
// ===== library: MasterCopy "BVS_Sensor" =====

FUNCTION_BLOCK "BVS_Sensor"   // FB52, SCL
TITLE = BVS_ID
{ S7_Optimized_Access := 'TRUE' }
AUTHOR : PD-ILS
FAMILY : Balluff
VERSION : 1.1
// Functionblock for BVS ID and BVS VS.
// Compatible with Profinet and IO-Link version.
   VAR_INPUT
      Init : Bool;   // Internal reset and initailisation of FB
      CommandStart : Bool;   // Start BVS command
      BVS_ResetError : Bool;   // Reset BVS errors
      BVS_Trigger : Bool;   // Trigger BVS
      Get_Results : Bool;   // Get BVS results
      HW_LADDR : HW_SUBMODULE;   // BVS hardware address
      Command : Int;   // 1=SwitchApp; 2=GetApp; 3=GetResult; 4=SetInput
      DB_Send : Int;   // Data block with BVS send data
      Offset_DBSend : Int;   // Offset send data
      DB_Receive : Int;   // Data block with BVS receive data
      Offset_DBReceive : Int;   // Offset receive data
      Data_Length : Int;   // Data length for set commando
      WD_Time : Time := T#120000ms;   // Watchdog of commandos
      PILen : UInt := 32;   // Input process data length
      PQLen : UInt := 32;   // Output process data length
   END_VAR
   VAR_OUTPUT
      Ready : Bool;   // Comamnd ready and FB ready
      BVS_WaitForTrigger : Bool;   // BVS waiting for Trigger
      BVS_ResultDataAvailable : Bool;   // BVS result ready
      BVS_Ready : Bool;   // BVS ready
      BVS_DeviceLocked : Bool;   // BVS is locked
      BVS_TriggerOverflowError : Bool;   // BVS warning overtriggerd
      BVS_ResultDataError : Bool;   // BVS warning result data error
      BVS_ReportError : Bool;   // BVS warning report error
      BVS_InputDataError : Bool;   // BVS warning input data error
      BVS_SystemError : Bool;   // BVS warning system error
      Error : Bool;   // Command or BVS Error
      ErrorNumber : Word;   // Error number
      ReceivedLength : Int;   // BVS received result buffer length
   END_VAR
   VAR
      PointerByte : Int;   // Pointer byte
      LengthByte : Int;   // Number of byte for set/get commando
      BytePerPageIn : Int;   // User bytes per page Out
      BytePerPageOut : Int;   // User bytes per page In
      TotalByte : Int;   // Over all byte data to be set/get
      LengOverhead : Int;   // Overhead length for get command
      StDataOffset : Int;   // Start Data Offset for set command
      HW_Init : Bool;   // Hardware adresses initialized
      GetCommandActive : Bool;   // Get commado activ
      SetCommandActive : Bool;   // Set commando active
      GComSend : Bool;   // Get Commando send
      ComDatEnd : Bool;   // Comand data transfered
      ToggleOld : Bool;   // Toggle bit last cycle
      FirstCycle : Bool;   // First command cycle
      IMP_Start : Bool;   // Rising edge Start
      IMP_ResetError : Bool;   // Rising edge Reset
      Cam_Reset : Bool;   // Start BVS reset
      ErrorIn : Bool;   // Error bit intern
      WD_TimerIn : Bool;   // Watchdog timer input
      WD_TimerQ : Bool;   // Watchdog timer output
      CO_WaitForTrigger : Bool;   // CAM Out - PLC In waiting for trigger BasAd[50]
      CO_ResultDataAvailable : Bool;   // CAM Out - PLC In result ready
      CO_R02 : Bool;   // CAM Out - PLC In reserved
      CO_R03 : Bool;   // CAM Out - PLC In simulation mode activated
      CO_R04 : Bool;   // CAM Out - PLC In reserved
      CO_Ready : Bool;   // CAM Out - PLC In ready
      CO_R06 : Bool;   // CAM Out - PLC In reserved
      CO_DeviceLocked : Bool;   // CAM Out - PLC In device locked
      CO_TriggerOverflow : Bool;   // CAM Out - PLC In error trigger overflow
      CO_ResultDataError : Bool;   // CAM Out - PLC In result data overwitten
      CO_ReportError : Bool;   // CAM Out - PLC In ftp report error
      CO_R13 : Bool;   // CAM Out - PLC In reserved
      CO_InputDataError : Bool;   // CAM Out - PLC Input data error
      CO_R15 : Bool;   // CAM Out - PLC In reserved
      CO_R16 : Bool;   // CAM Out - PLC In reserved
      CO_SystemError : Bool;   // CAM Out - PLC In system error
      CO_R20 : Bool;   // CAM Out - PLC In reserved
      CO_JobStartAA : Bool;   // CAM Out - PLC In job start
      CO_JobEndAE : Bool;   // CAM Out - PLC In job end
      CO_JobErrorAF : Bool;   // CAM Out - PLC In job error
      CO_R24 : Bool;   // CAM Out - PLC In reserved
      CO_ToggleOut : Bool;   // CAM Out - PLC In toggle out
      CO_OutArea : Array[0..#OutBuSi] of Byte;   // CAM Out - PLC In data area
      CI_AV_JobStart : Bool;   // PLC Out - CAM In job start
      CI_Trigger : Bool;   // PLC Out - CAM In trigger
      CI_ResetError : Bool;   // PLC Out - CAM In reset error
      CI_R03 : Bool;   // PLC Out - CAM In reserved
      CI_R04 : Bool;   // PLC Out - CAM In reserved
      CI_R05 : Bool;   // PLC Out - CAM In reserved
      CI_ToggleIn : Bool;   // PLC Out - CAM In toggle in
      CI_R07 : Bool;   // PLC Out - CAM In reserved
      CI_InLengInt : Int;   // PLC Out - CAM In length int
      CI_InArea : Array[0..#InBuSi] of Byte;   // PLC Out - CAM In input area
      OldCyComState : Word;   // Commando state last cycle
      WD_Timer : TON_TIME;   // Watchdog timer TON
      PIaddr : UDInt;   // Input address
      PIcount : UInt;   // Input length
      PQaddr : UDInt;   // Output address
      PQcount : UInt;   // Output address
      RetVal_ModulDiag : Int;   // Return value modul diagnosis
      RetVal_RD_Addr : Int;   // Return value read address
      RetVal_RD_DP : Int;   // Return value read input data
      RetVal_WR_DP : Int;   // Return value write output data
      RetVal_Get_ErrID : Word;   // Return value get error ID
      R_TRIG_ResetError : R_TRIG;   // R Trigger reset warning
      R_TRIG_CamTrg : R_TRIG;   // R Trigger BVS trigger
      R_TRIG_Start : R_TRIG;   // R Trigger BVS start
      ErrorCode : DWord;   // Internal BVS error code
      CNT_Diag : UInt;   // CNT_Modul Diag
      Diag_Out : DWord;   // Modul Diag
   END_VAR
   VAR_TEMP
      tError : Word;   // temp error buffer
      tLoop : DInt;   // temp loopcounter
   END_VAR
   VAR CONSTANT
      InBuSi : Int := 127;   // maximum size input buffer
      OutBuSi : Int := 127;   // maximum size output buffer
      ST_DATOFFSET : Int := 3;   // First DataOffset for set commands
   END_VAR
BEGIN
   //=============================================================================
   //Balluff GmbH
   //(c)Copyright (2024) All Rights Reserved
   //-----------------------------------------------------------------------------
   //Library: BalluffVision
   //Tested with: CPU 1214C V4.1
   //Engineering: TIA Portal V13 SP1 
   //Restrictions: -
   //Requirements: PLC (S7-1200 / S7-1500)
   //Functionality: Boolean BVS functions, BVS Commandos
   //-----------------------------------------------------------------------------
   //Change log table:
   //Version  Date       Expert in charge      Changes applied
   //00.01.00 30.11.2022 Balluff GmbH PD-ILS   First created with TIA V13 SP1
   //00.01.10 30.01.2024 Balluff GmbH PD-ILS   FB name changed, buffer enlarged
   //=============================================================================
   //
   (*
   Disclaimer of Liability
   **********************
   The demo function block is free of charge and is a universal application 
   example.
   This demo function block shall help program and configure PLC applications and 
   shall provide possible solutions.
   The user is not entitled to claim for warranty, error correction and updates. 
   In 
   particular there is excluded any claims against Balluff GmbH for damages that 
   might result from the use of this demo program. Excluded from this limitation 
   of 
   liability shall be (a) those damages that are based on injury to life, limb or 
   health, (b) a liability according to the Produkthaftungsgesetz (German Product 
   Liability Law) and (c) cases of willful intent.
   Please check if the function block is intended for your application before 
   adapting it in plants and machineries.
   By using the S7 sample, made available free of charge you accept the limitation 
   of 
   warranty and liability!

   Haftungsausschluss:
   *********************
   Der hier kostenlos verfügbare DEMO-Baustein ist ein allgemeingültiges 
   Anwendungsbeispiel. Dieser DEMO-Baustein soll bei der Programmierung und 
   Projektierung von SPS-Anwendungen unterstützen und Lösungsansätze aufzeigen. 
   Ein Anspruch auf Gewährleistung, Fehlerbeseitigung und Update besteht für den 
   Anwender nicht. Die BALLUFF GmbH schließt insbesondere jegliche Haftung für 
   Schäden, die durch den Einsatz dieses DEMO-Bausteins entstehen, ausdrücklich 
   aus! Diese Haftungsbeschränkung gilt nicht bei Verletzungen des Lebens, des 
   Körpers oder der Gesundheit, bei der Haftung nach dem Produkthaftungsgesetz und 
   bei vorsätzlichen Pflichtverletzungen. 
   Prüfen Sie vor dem Einsatz in Anlagen und Maschinen, ob der hier 
   bereitgestellte 
   DEMO Baustein für Ihre Anwendung nutzbar ist!
   Mit dem Einsatz des hier kostenlos vorgelegten S7-Beispiel erkennen Sie die 
   Gewährleistungs- und Haftungsbegrenzung an!
   *)
   //-----------------------------------------------------------------------------
   //FB Init
   //-----------------------------------------------------------------------------
   IF #Init THEN
       #Ready := TRUE;
       #HW_Init := FALSE;
       #GetCommandActive := FALSE;
       #SetCommandActive := FALSE;
       #GComSend := FALSE;
       #ToggleOld := FALSE;
       #FirstCycle := FALSE;
       #ComDatEnd := False;
       #Error := FALSE;
       #ErrorIn := FALSE;
       #CI_AV_JobStart := FALSE;
       #CI_Trigger := FALSE;
       #CI_ResetError := false;
       #PointerByte := 0;
       #BytePerPageIn := 0;
       #BytePerPageOut := 0;
       #TotalByte := 0;
       #ReceivedLength := 0;
       #ErrorNumber := 0;
       #CO_OutArea[0] := 0;
       #CO_OutArea[1] := 0;
       #CO_OutArea[2] := 0;
       #BVS_Ready := FALSE;
   END_IF;
   //-----------------------------------------------------------------------------
   // Read modul states
   //-----------------------------------------------------------------------------
   #RetVal_ModulDiag := GET_DIAG(MODE := 0, LADDR := #HW_LADDR, CNT_DIAG => #CNT_Diag, DIAG := #Diag_Out);

   //-----------------------------------------------------------------------------
   // Reading PI/PQ addr and data length
   //-----------------------------------------------------------------------------
   IF NOT #HW_Init THEN
     #RetVal_RD_Addr := RD_ADDR(LADDR := #HW_LADDR , PIADDR => #PIaddr, PICount => #PIcount,
                                  PQADDR => #PQaddr, PQCount => #PQcount);
       #HW_Init := TRUE;
       // Overwrite PI and PO Lenght with lenth from FB input
       #PIcount := #PILen;
       #PQcount := #PQLen;
   END_IF;
   //-----------------------------------------------------------------------------
   // Cyclic read cam input if HW init done
   //----------------------------------------------------------------------------- 
   IF #HW_Init THEN
     #RetVal_RD_DP := DPRD_DAT(LADDR := #HW_LADDR, RECORD => #CO_OutArea);
   END_IF;

   IF #RetVal_RD_DP <> 0 THEN
     FOR  #tLoop := 0 TO #OutBuSi DO
       #CO_OutArea[#tLoop] := 0;
     END_FOR;
   END_IF;

   IF #Init THEN
     GOTO JobReset;
   END_IF;
   //-----------------------------------------------------------------------------
   // Move input bytes to static bits
   //  CO == Camera Outputs
   //-----------------------------------------------------------------------------
   // Byte 0 - Product Status Bits
   #CO_WaitForTrigger := #CO_OutArea[0].%X0;
   #CO_ResultDataAvailable := #CO_OutArea[0].%X1;
   #CO_R02 := #CO_OutArea[0].%X2;
   #CO_R03 := #CO_OutArea[0].%X3;
   #CO_R04 := #CO_OutArea[0].%X4;
   #CO_Ready := #CO_OutArea[0].%X5;
   #CO_R06 := #CO_OutArea[0].%X6;
   #CO_DeviceLocked := #CO_OutArea[0].%X7;
   //Byte 1 - Error Signals
   #CO_TriggerOverflow := #CO_OutArea[1].%X0;
   #CO_ResultDataError := #CO_OutArea[1].%X1;
   #CO_ReportError := #CO_OutArea[1].%X2;
   #CO_R13 := #CO_OutArea[1].%X3;
   #CO_InputDataError := #CO_OutArea[1].%X4;
   #CO_R15 := #CO_OutArea[1].%X5;
   #CO_R16 := #CO_OutArea[1].%X6;
   #CO_SystemError := #CO_OutArea[1].%X7;

   //-----------------------------------------------------------------------------
   // Move status-/warnbits to FB output 
   //-----------------------------------------------------------------------------
   #BVS_ResultDataAvailable := #CO_ResultDataAvailable;
   #BVS_WaitForTrigger := #CO_WaitForTrigger;
   #BVS_Ready := #CO_Ready;
   #BVS_DeviceLocked := #CO_DeviceLocked;
   #BVS_TriggerOverflowError := #CO_TriggerOverflow;
   #BVS_ResultDataError := #CO_ResultDataError;
   #BVS_ReportError := #CO_ReportError;
   #BVS_InputDataError := #CO_InputDataError;
   #BVS_SystemError := #CO_SystemError;

   //-----------------------------------------------------------------------------
   // Comapre bitheader
   //-----------------------------------------------------------------------------
   IF #CO_OutArea[2] <> #CO_OutArea[#PIcount - 1] THEN
     RETURN;
   END_IF;
   //Byte 2 - Bit Header
   #CO_R20 := #CO_OutArea[2].%X0;
   #CO_JobStartAA := #CO_OutArea[2].%X1;
   #CO_JobEndAE := #CO_OutArea[2].%X2;
   #CO_JobErrorAF := #CO_OutArea[2].%X3;
   #CO_ToggleOut := #CO_OutArea[2].%X5;

   //-----------------------------------------------------------------------------
   // Check camera error bit
   //-----------------------------------------------------------------------------
   IF #CO_JobErrorAF AND NOT #ErrorIn THEN
     #tError := #CO_OutArea[3];
     GOTO Error;
   END_IF;

   //-----------------------------------------------------------------------------
   // Reset camera errors
   //-----------------------------------------------------------------------------
   #R_TRIG_ResetError(CLK:=#BVS_ResetError,
                   Q=>#IMP_ResetError);
   IF #IMP_ResetError THEN
       #Error := FALSE;
       #ErrorIn := FALSE;
       #ErrorNumber := 0;
       #CI_ResetError := TRUE;
   END_IF;

   IF NOT #BVS_ResetError
     THEN
       #CI_ResetError := FALSE;
   END_IF;

   //-----------------------------------------------------------------------------
   // Control boolean camera signals
   //-----------------------------------------------------------------------------
   #R_TRIG_CamTrg(CLK:=#BVS_Trigger);

   IF #R_TRIG_CamTrg.Q THEN
     #CI_Trigger := TRUE;
   END_IF;

   IF  NOT #BVS_Trigger THEN
     #CI_Trigger := FALSE;
   END_IF;

   //-----------------------------------------------------------------------------
   // Move  FB input to processdata output
   //-----------------------------------------------------------------------------
   #CI_InArea[0].%X0 := #CI_AV_JobStart;
   #CI_InArea[0].%X1 := #CI_Trigger;
   #CI_InArea[0].%X2 := #CI_ResetError;
   #CI_InArea[0].%X6 := #CI_ToggleIn;

   //-----------------------------------------------------------------------------
   // FB ready output 
   #Ready := ( #BVS_Ready 
             AND NOT #GetCommandActive 
             AND NOT #SetCommandActive 
             AND NOT #CO_JobStartAA 
             AND NOT #CO_JobEndAE);

   //-----------------------------------------------------------------------------
   // Command Start
              #R_TRIG_Start(CLK := #CommandStart OR #Get_Results,
                 Q => #IMP_Start);

   //-----------------------------------------------------------------------------
   // Generate error timeout
   //-----------------------------------------------------------------------------
   #WD_TimerIn := #SetCommandActive OR #GetCommandActive;

   #WD_Timer(IN := #WD_TimerIn,
             PT := #WD_Time,
             Q => #WD_TimerQ);

   IF #WD_TimerQ THEN
       #tError := w#16#30;
       GOTO Error;
   END_IF;

   //-----------------------------------------------------------------------------
   // Check HW/Profinet Error when start is set
   //-----------------------------------------------------------------------------
   IF #IMP_Start THEN
     IF #RetVal_RD_Addr <> 0 THEN
       #tError := w#16#40; //Error read address
       GOTO Error;
     END_IF;

     IF #RetVal_RD_DP <> 0 THEN
       #tError := w#16#41; //Error read input data
       GOTO Error;
     END_IF;

     IF #RetVal_WR_DP <> 0 THEN
       #tError := w#16#42; //Error read output data
       GOTO Error;
     END_IF;
   END_IF;

   //-----------------------------------------------------------------------------
   // Generate error data length
   //-----------------------------------------------------------------------------
   IF #IMP_Start AND
       (#Data_Length < 0) THEN
       #tError := w#16#32;
       GOTO Error;
   END_IF;

   //-----------------------------------------------------------------------------
   // Check controll- bits change - data output
   //-----------------------------------------------------------------------------
   IF #CI_InArea[0] <> #OldCyComState AND NOT #IMP_Start THEN
     GOTO DataOutput;
   END_IF;
   //=============================================================================
   //
   // Camera commandos
   //
   //=============================================================================

   //-----------------------------------------------------------------------------
   // Goto FB end if no job active
   //-----------------------------------------------------------------------------
   IF (NOT #GetCommandActive AND
       NOT #SetCommandActive AND
      (NOT #IMP_Start OR NOT #Ready)) THEN 
       RETURN;
   END_IF;

   IF #ComDatEnd THEN  // Check Get or Set
     GOTO CheckHsAck; //CommandEnd;
   ELSIF #GetCommandActive THEN
     GOTO GetCommand;
   ELSIF #SetCommandActive THEN
     GOTO SetCommand;
   END_IF;

   //-----------------------------------------------------------------------------
   // Initialize Command
   //-----------------------------------------------------------------------------
   #CI_InArea[2] := 0;
   #CI_InArea[3] := 0;

   IF #Get_Results THEN
     #GetCommandActive := TRUE;
     #CI_InArea[1] := 3;
     #CI_InLengInt := 0;
     #LengOverhead := 3;
   ELSE

     CASE #Command OF
       1: // Switch Application
         #SetCommandActive := TRUE;
         #CI_InArea[1] := 1;
         #TotalByte := 4;
         #CI_InLengInt := 4;
       2:  // Get Application ID
         #GetCommandActive := TRUE;
         #CI_InArea[1] := 2;
         #CI_InLengInt := 0;
         #LengOverhead := 3;
       3:  // Get Results
         #GetCommandActive := TRUE;
         #CI_InArea[1] := 3;
         #CI_InLengInt := 0;
         #LengOverhead := 3;
       4:  // Set Inputs       
         #SetCommandActive := TRUE;
         #CI_InArea[1] := 4;
         #TotalByte := #Data_Length;
         #CI_InLengInt := #Data_Length;
       6:  // Get Date and Time 
         #GetCommandActive := TRUE;
         #CI_InArea[1] := 6;
         #CI_InLengInt := 0;
         #LengOverhead := 3;
       7:  // Set Date and Time      
         #SetCommandActive := TRUE;
         #CI_InArea[1] := 7;
         #TotalByte := 7 + #ST_DATOFFSET;
         #CI_InLengInt := 7;
       ELSE
         #tError := w#16#31;
         GOTO Error;
     END_CASE;
   END_IF;

   //-----------------------------------------------------------------------------
   // At 1st command step:
   // Calculate transmission data length fix bytes + bitheader
   // Delete output signals
   // Notice TO Bit
   //-----------------------------------------------------------------------------
   #BytePerPageIn := UDINT_TO_INT(#PIcount - 4);
   #BytePerPageOut := UDINT_TO_INT(#PQcount - 2);

   #FirstCycle := TRUE;
   #Ready := FALSE;
   #ErrorNumber := 0;
   #Error := FALSE;
   #ErrorIn := FALSE;
   #tError := 0;
   #GComSend := FALSE;
   #ReceivedLength := 0;
   #ToggleOld := #CO_ToggleOut;
   #CI_AV_JobStart := TRUE;

   IF NOT #SetCommandActive THEN
       GOTO GetCommand;
   END_IF;

   //-----------------------------------------------------------------------------
   // Set command, move data from "DB_Send" to camera
   //-----------------------------------------------------------------------------
   SetCommand: ;

   IF NOT #FirstCycle  
       AND ((#ToggleOld AND #CO_ToggleOut)
       OR (NOT #ToggleOld AND NOT #CO_ToggleOut)
       OR  NOT #CO_JobStartAA)
     THEN
       RETURN;
   END_IF;

   IF #FirstCycle THEN
     #PointerByte := #Offset_DBSend;
     #StDataOffset := #ST_DATOFFSET;
     #CI_InArea[2] := INT_TO_BYTE(SHR(IN := #CI_InLengInt, N := 8)); 
     #CI_InArea[3] := INT_TO_BYTE(#CI_InLengInt); 
   END_IF;

   IF #TotalByte <= #BytePerPageOut - #StDataOffset THEN
     #LengthByte := #TotalByte;
   ELSE
     #LengthByte := #BytePerPageOut - #StDataOffset;
   END_IF;

   FOR #tLoop := 0 TO #LengthByte - 1 DO 
     #CI_InArea[1 + #tLoop + #StDataOffset] := PEEK(area := 16#84,
                                      dbNumber := #DB_Send,
                                      byteOffset := #PointerByte + #tLoop);
     END_FOR;

   GOTO CommandEnd;

   GetCommand:;
   //-----------------------------------------------------------------------------
   // Get command
   // Send get commando goto Data output in first cycle 
   // 
   //-----------------------------------------------------------------------------
   IF #FirstCycle AND NOT #GComSend THEN
     #GComSend := TRUE;
     GOTO DataOutput;
   END_IF;

   IF #FirstCycle AND #CI_InArea[1] <> #CO_OutArea[3] // Check result code at 1st cycl 
     AND NOT #CO_JobStartAA
     OR NOT #CO_JobEndAE 
   THEN
     RETURN;
   END_IF;

   IF NOT #FirstCycle
     AND ((#ToggleOld AND #CO_ToggleOut)
     OR (NOT #ToggleOld AND NOT #CO_ToggleOut))
   THEN
     RETURN;
   END_IF;

   //-----------------------------------------------------------------------------
   // Read camera length byte at 1st cycle
   // move data from camera to "DB_Receive"
   //  
   //----------------------------------------------------------------------------- 
   IF #FirstCycle THEN

     #TotalByte := BYTE_TO_INT(#CO_OutArea[5]) +
     SHL(IN := BYTE_TO_INT(#CO_OutArea[4]), N := 8)+
     #LengOverhead;

     #PointerByte := #Offset_DBReceive;

     IF (#TotalByte < 0) THEN
       #tError := 16#32;
       GOTO Error;
     END_IF;

     #ReceivedLength := #TotalByte;

   END_IF; // End_IF First Cycle

   IF #TotalByte <= #BytePerPageIn THEN
     #LengthByte := #TotalByte;
    ELSE
     #LengthByte := #BytePerPageIn;
   END_IF;

   FOR #tLoop := 0 TO #LengthByte - 1 DO
     POKE(area := 16#84,
          dbNumber := #DB_Receive,
          byteOffset := #PointerByte + #tLoop,
          value := #CO_OutArea[3 + #tLoop]);
   END_FOR;

   CommandEnd:;

   //-----------------------------------------------------------------------------
   // Get and Set Command End
   //----------------------------------------------------------------------------- 
   IF NOT #ComDatEnd THEN
     #TotalByte := #TotalByte - #LengthByte;
     #PointerByte := #PointerByte + #LengthByte;
   END_IF;

   IF #TotalByte <= 0 THEN
     #ComDatEnd := TRUE;
   END_IF;

   IF (#GetCommandActive AND NOT #ComDatEnd) OR
     (NOT #FirstCycle AND #SetCommandActive) THEN
     #CI_ToggleIn := NOT #CI_ToggleIn;
   END_IF;

   #ToggleOld := #CO_ToggleOut;
   #FirstCycle := FALSE;
   #StDataOffset := 0;
   CheckHsAck:;

   IF (#CO_JobStartAA AND #CO_JobEndAE AND #ComDatEnd) THEN 
       #ComDatEnd := FALSE;
       #GetCommandActive := FALSE;
       #SetCommandActive := FALSE;
       #CI_AV_JobStart := FALSE;
       #CI_ToggleIn := FALSE;
       #ToggleOld := FALSE;
   END_IF;

   //-----------------------------------------------------------------------------
   // Data output fieldbus
   //-----------------------------------------------------------------------------
   DataOutput:;
   // Move bits to byte
   #CI_InArea[0].%X0 := #CI_AV_JobStart;
   #CI_InArea[0].%X1 := #CI_Trigger;
   #CI_InArea[0].%X2 := #CI_ResetError;
   #CI_InArea[0].%X6 := #CI_ToggleIn ;
   #CI_InArea[#PQcount - 1] := #CI_InArea[0];
   #OldCyComState := #CI_InArea[0];

   //-----------------------------------------------------------------------------
   // cyclic write plc output to cam input
   //-----------------------------------------------------------------------------
   IF #HW_Init  THEN
     #RetVal_WR_DP := DPWR_DAT(LADDR := #HW_LADDR, RECORD := #CI_InArea);
   END_IF;
   #RetVal_Get_ErrID := GET_ERR_ID();

   IF #RetVal_Get_ErrID <> 0
     AND NOT #Init
     AND NOT #ErrorIn THEN
     #tError := 16#43;
     GOTO Error;
   END_IF;

   RETURN; // FB End
   //-----------------------------------------------------------------------------
   // Error output
   //-----------------------------------------------------------------------------
   Error: ;
     #ErrorNumber := #tError;
     #Ready := FALSE;
     #Error := TRUE;
     #ErrorIn := TRUE;

   JobReset: ;
     #GetCommandActive := FALSE;
     #SetCommandActive := FALSE;
     #CI_AV_JobStart := FALSE;
     #CI_ToggleIn := FALSE;
     #ComDatEnd := FALSE;
     #ToggleOld := FALSE;
     GOTO DataOutput;
END_FUNCTION_BLOCK